// TIA Portal V16 export
// export: Created 2023-03-29T11:03:48.1346201Z, ExportSetting WithDefaults, DisplayName Totally Integrated Automation Portal, DisplayVersion V16 Update 6, DisplayName TIA Portal Version Control Interface, DisplayVersion V16 Update 2, DisplayName TIA Portal Openness, DisplayVersion V16 Update 6, DisplayName STEP 7 Professional, DisplayVersion V16 Update 6, DisplayName STEP 7 Safety, DisplayVersion V16, DisplayName WinCC Advanced, DisplayVersion V16 Update 6
TYPE "typeModbusSlave"
// stored: IsFailsafeCompliant false
   STRUCT
      NDR : Bool := FALSE;   // New data ready: 1: Indicates that data has been read by the Modbus master No new data
      mbAddr : UInt;   // Station address of the Modbus slave (address range: 0 to 255)
      done : Bool := FALSE;   // Boolean indicating completion without error
      dr : Bool := FALSE;   // Read data: 0: No data read1: Indicates that data has been read by the Modbus master
      error : Bool := FALSE;   // Boolean indicating completion with error
      status : Word := W#16#0;   // Status or error code of the completed operation
      errorStatus : Word := W#16#0;   // Error code of the faulty operation
   END_STRUCT;
END_TYPE
